# EPICS autosave request: iocBoot/iocMeasComp/auto_settings.req
file "C9513_settings.req", P=C9513:
file "1608G_settings.req", P=1608G:
